PROGRAM MAIN
VAR
    Machine : MachineModule('Machine 1');
    Machine_HMI : PackMLStatemachine_HMI('Machine 1 HMI', Machine);
END_VAR

Machine.CyclicLogic();
Machine_HMI.CyclicLogic();

END_PROGRAM

(* stored: Version 1.1.0.1, ProductVersion 3.1.4026.18
   POU MAIN: Id {8644c25d-c61e-485a-a0b5-43a6501af7bc}, SpecialFunc None *)
